TYPE ST_Test :
STRUCT
	rTest	: REAL;
	iTest	: INT;
	bTest	: BOOL;
END_STRUCT
END_TYPE

(* stored: Version 1.1.0.1, ProductVersion 3.1.4024.2
   DUT ST_Test: Id {f92d63c4-89e9-4803-9561-72ce61ca8969} *)
